// LS Electric XG5000 project: 24.실린더 1개, 모터 2개 제어
// PLC NewPLC
// module base 0 slot 0: 입출력 모듈:XBM-DN/DP32HP (DC 24V입력/TR 출력, 32점)
// module base 0 slot 2: 입력 모듈:XBE-DC08A (DC 24V 입력, 8점 (전류소스 싱크공용))

PROGRAM NewProgram (task: 스캔 프로그램)

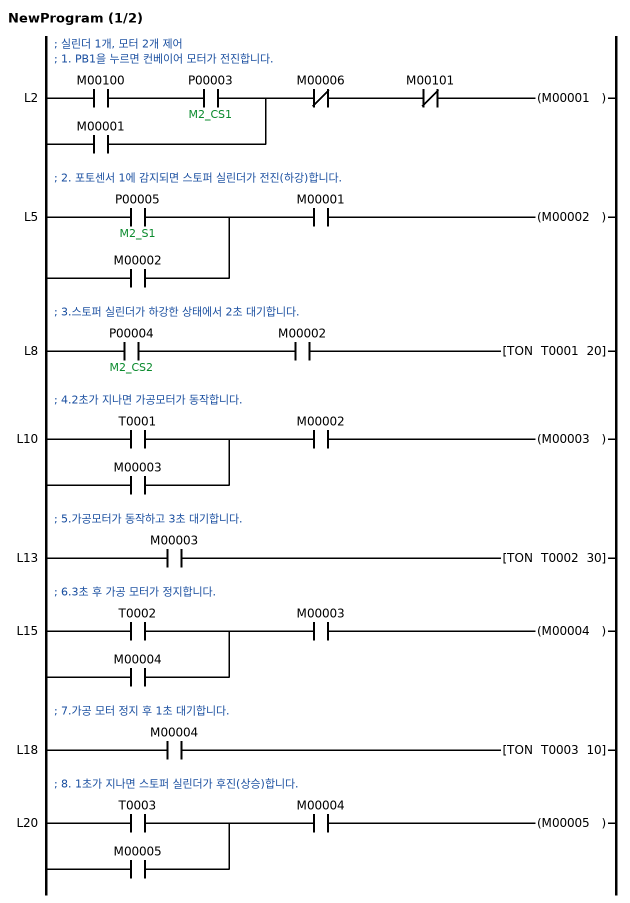
// 실린더 1개, 모터 2개 제어
// 1. PB1을 누르면 컨베이어 모터가 전진합니다.
; L2
LOAD      M00100
AND       P00003	// M2_CS1
OR        M00001
AND NOT   M00006
AND NOT   M00101
OUT       M00001
// 2. 포토센서 1에 감지되면 스토퍼 실린더가 전진(하강)합니다.
; L5
LOAD      P00005	// M2_S1
OR        M00002
AND       M00001
OUT       M00002
// 3.스토퍼 실린더가 하강한 상태에서 2초 대기합니다.
; L8
LOAD      P00004	// M2_CS2
AND       M00002
TON       T0001 20
// 4.2초가 지나면 가공모터가 동작합니다.
; L10
LOAD      T0001
OR        M00003
AND       M00002
OUT       M00003
// 5.가공모터가 동작하고 3초 대기합니다.
; L13
LOAD      M00003
TON       T0002 30
// 6.3초 후 가공 모터가 정지합니다.
; L15
LOAD      T0002
OR        M00004
AND       M00003
OUT       M00004
// 7.가공 모터 정지 후 1초 대기합니다.
; L18
LOAD      M00004
TON       T0003 10
// 8. 1초가 지나면 스토퍼 실린더가 후진(상승)합니다.
; L20
LOAD      T0003
OR        M00005
AND       M00004
OUT       M00005

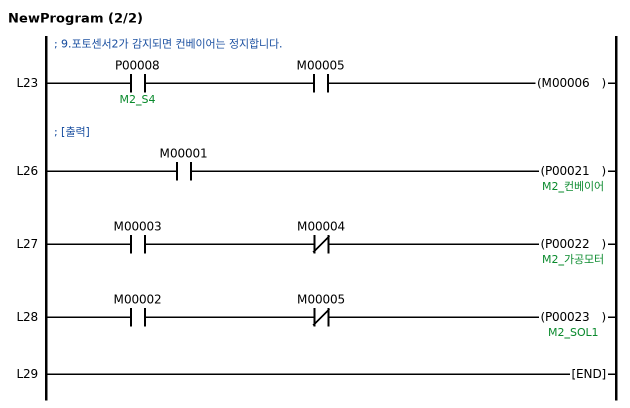
// 9.포토센서2가 감지되면 컨베이어는 정지합니다.
; L23
LOAD      P00008	// M2_S4
AND       M00005
OUT       M00006
// [출력]
; L26
LOAD      M00001
OUT       P00021	// M2_컨베이어
; L27
LOAD      M00003
AND NOT   M00004
OUT       P00022	// M2_가공모터
; L28
LOAD      M00002
AND NOT   M00005
OUT       P00023	// M2_SOL1
; L29
END

VARIABLES AND COMMENTS (devices not used above)
P00080	BIT	PB1
P00081	BIT	PB2
P00029	BIT	PL2_YELLOW
P00028	BIT	PL1_GREEN
P00083	BIT	PB4
P00082	BIT	PB3
P0002A	BIT	PL3_RED
P00020	BIT	M1_SOL1
P00000	BIT	M1_CS1
P00001	BIT	M1_CS2
P00002	BIT	M1_S1